Universal Robots PolyScope program: d02_cycle.urp

Program d02_cycle (installation=default directory=/programs createdIn=5.9.1.1031110 lastSavedIn=5.9.1.1031110 robotSerialNumber=20195501059)
Calibrated DH parameters: a=[0.000146, -0.418764, -0.053981, 0.000058, -0.000023, 0]; d=[0.162545, 37.319448, -206.067439, 168.881546, 0.09955, 0.099464]; alpha=[1.57004, -0.001979, 0.002304, 1.570607, -1.57066, 0]; deltaTheta=[0, -0.174616, -1.258233, 1.432844, -0.000001, 0]
BeforeStart
  URCap Gripper Activate (Robotiq_Grippers, Robotiq Inc.) dataModel(ResetAndActivateKey=false)
Robot Program (runOnlyOnce=true)
  Call d02_home
  Call d02_amp_off
  Call d02_unplug
  Call d02_replug
  Call d02_amp_on
  Call d02_home
SubProgram -> d02_home
SubProgram -> d02_amp_off
SubProgram -> d02_amp_on
SubProgram -> d02_unplug
SubProgram -> d02_replug
SubProgram d02_home (keepSynchronizedWithDisk=true) programFile=/programs/d02_home.urp
  URCap Gripper Activate (Robotiq_Grippers, Robotiq Inc.) dataModel(ResetAndActivateKey=false)
  URCap Gripper (Robotiq_Grippers, Robotiq Inc.) dataModel(position=65.0, force=100.0, speed=100.0, positionInDouble=65.0, forceInDouble=100.0, speedInDouble=100.0, slaveIds=[9], blocking=true)
  URCap Gripper (Robotiq_Grippers, Robotiq Inc.) dataModel(position=100.0, force=100.0, speed=100.0, positionInDouble=100.0, forceInDouble=100.0, speedInDouble=100.0, slaveIds=[9], blocking=false)
  MoveJ speed 60 deg/s, acceleration 80 deg/s^2 (useActiveTCP=true) feature=Base
    Waypoint Waypoint (Variable): variable(featureName=d02_home_p)
SubProgram d02_amp_off (keepSynchronizedWithDisk=true) programFile=/programs/d02_amp_off.urp
  URCap Gripper (Robotiq_Grippers, Robotiq Inc.) dataModel(position=100.0, force=100.0, speed=100.0, positionInDouble=100.0, forceInDouble=100.0, speedInDouble=100.0, slaveIds=[9], blocking=false)
  MoveL speed 250 mm/s, acceleration 1200 mm/s^2 (useActiveTCP=true) feature=Base
    Waypoint Waypoint (Variable): variable(featureName=d02_amp_sw_p)
    URCap Zero FT Sensor (Robotiq_Copilot, Robotiq Inc.) dataModel(NodeInitializedKey=true, WaitForSteadyWrenchOptionKey=true)
    URCap Force Control (Robotiq_Copilot, Robotiq Inc.) dataModel(NodeInitializedKey=true, force_x=0, force_y=0, force_mx=0, force_my=0, force_mz=0, limit_x_neg=-100, limit_y_neg=-100, limit_z_neg=-100, limit_x_pos=100, limit_y_pos=100, limit_z_pos=100, limit_mx_neg=-20, limit_my_neg=-20, limit_mz_neg=-20, limit_mx_pos=20, limit_my_pos=20, limit_mz_pos=20, ft_control_mx=false, ft_control_my=false, ft_control_mz=false, stiffness_x=100, stiffness_y=100, stiffness_z_position=100, stiffness_mx=100, stiffness_my=100, stiffness_mz=100, force_z=20, ft_control_y=false, ft_control_x=false, HackTriggeringContributionIsDefinedMethodKey=true, TranslatableFeatureKey=1, adaptive_stiffness=true, ft_control_z=true, is_force_control_about_actual_position=true)
      Wait Sleep waitTime=2
    Waypoint Waypoint (Variable): variable(featureName=d02_amp_sw_p)
SubProgram d02_unplug (keepSynchronizedWithDisk=true) programFile=/programs/d02_unplug.urp
  MoveL speed 250 mm/s, acceleration 1200 mm/s^2 (useActiveTCP=true) feature=Base
    Waypoint Waypoint (Variable): variable(featureName=d02_plug_p)
    URCap Gripper (Robotiq_Grippers, Robotiq Inc.) dataModel(position=100.0, force=100.0, speed=100.0, positionInDouble=100.0, forceInDouble=100.0, speedInDouble=100.0, slaveIds=[9], blocking=false)
    MoveDirectionNode (selectedDirection=ZPlus toolParams=0.02, 0.8) feature=Joint_6_name
      Until TOOL_CONTACT_DETECTION (allowActions=true retraction=0.001 decelerationAcceleration=3 decelerationAngularAcceleration=34.906585)
        URCap Gripper (Robotiq_Grippers, Robotiq Inc.) dataModel(position=65.0, force=100.0, speed=100.0, positionInDouble=65.0, forceInDouble=100.0, speedInDouble=100.0, slaveIds=[9], blocking=true)
        MoveDirectionNode (selectedDirection=ZPlus toolParams=0.05, 0.8) feature=Joint_6_name
          Until DISTANCE (allowActions=false deceleration=3 distanceNodeType=STOP) Distance=0.02; motionParameters(blendRadius=0)
        URCap Gripper (Robotiq_Grippers, Robotiq Inc.) dataModel(position=100.0, force=100.0, speed=100.0, positionInDouble=100.0, forceInDouble=100.0, speedInDouble=100.0, slaveIds=[9], blocking=true)
        MoveL speed 25 mm/s, acceleration 1200 mm/s^2 (useActiveTCP=true) feature=Base
          Waypoint Pull (Relative): relativeFromPosition TCP in base x=108.075 y=-582.031 z=19.139 mm, rx=-2.2457 ry=-2.1683 rz=0.0242 rad; joints [88.128, -64.848, 105.271, -130.26, 268.593, 90.173] deg; TCP offset x=0 y=0 z=174 mm, rx=0 ry=0 rz=0 rad; TCP in base x=109.536 y=-542.231 z=19.13 mm, rx=-2.2458 ry=-2.1682 rz=0.0241 rad; joints [88.149, -69.075, 111.89, -132.649, 268.605, 90.202] deg
      Until DISTANCE (allowActions=true deceleration=3 distanceNodeType=STOP) Distance=0.02; motionParameters(blendRadius=0)
        Waypoint Waypoint (Variable): variable(featureName=d02_plug_p)
SubProgram d02_replug (keepSynchronizedWithDisk=true) programFile=/programs/d02_replug.urp
  URCap Insertion (Robotiq_Copilot, Robotiq Inc.) dataModel(NodeInitializedKey=true)
    URCap Zero FT Sensor (Robotiq_Copilot, Robotiq Inc.) dataModel(NodeInitializedKey=true, WaitForSteadyWrenchOptionKey=false)
    URCap Linear (Robotiq_Copilot, Robotiq Inc.) dataModel(NodeInitializedKey=true, fb_exit_insertion=false, fb_max_distance=50.0, fb_speed=10.0, fb_force=40.0, fbDirection=X-); state(isChildrenLocked=true)
      URCap On error (Robotiq_Copilot, Robotiq Inc.)
        'Sequence if maximum distance is reached'
        Halt
    URCap Gripper (Robotiq_Grippers, Robotiq Inc.) dataModel(position=65.0, force=100.0, speed=100.0, positionInDouble=65.0, forceInDouble=100.0, speedInDouble=100.0, slaveIds=[9], blocking=true)
    MoveL speed 250 mm/s, acceleration 1200 mm/s^2 (useActiveTCP=true) feature=Base
      MoveDirectionNode (selectedDirection=ZMinus) feature=Joint_6_name
        Until DISTANCE (allowActions=false deceleration=3 distanceNodeType=STOP) Distance=0.025; motionParameters(blendRadius=0)
SubProgram d02_amp_on (keepSynchronizedWithDisk=true) programFile=/programs/d02_amp_on.urp
  URCap Gripper (Robotiq_Grippers, Robotiq Inc.) dataModel(position=100.0, force=100.0, speed=100.0, positionInDouble=100.0, forceInDouble=100.0, speedInDouble=100.0, slaveIds=[9], blocking=false)
  MoveL speed 250 mm/s, acceleration 1200 mm/s^2 (useActiveTCP=true) feature=Base
    Waypoint Waypoint (Variable): variable(featureName=d02_amp_sw_p)
    MoveDirectionNode (selectedDirection=ZPlus toolParams=0.01, 0.8) feature=Joint_6_name
      Until TOOL_CONTACT_DETECTION (allowActions=false retraction=0 decelerationAcceleration=3 decelerationAngularAcceleration=34.906585)
    URCap Gripper (Robotiq_Grippers, Robotiq Inc.) dataModel(position=75.29411764705883, force=100.0, speed=100.0, positionInDouble=75.29411764705883, forceInDouble=100.0, speedInDouble=100.0, slaveIds=[9], blocking=true)
    MoveDirectionNode (selectedDirection=ZPlus toolParams=0.01, 0.8) feature=Joint_6_name
      Until DISTANCE (allowActions=false deceleration=3 distanceNodeType=STOP) Distance=0.01; motionParameters(blendRadius=0)
    URCap Gripper (Robotiq_Grippers, Robotiq Inc.) dataModel(position=100.0, force=100.0, speed=100.0, positionInDouble=100.0, forceInDouble=100.0, speedInDouble=100.0, slaveIds=[9], blocking=true)
    URCap Force Control (Robotiq_Copilot, Robotiq Inc.) dataModel(NodeInitializedKey=true, force_x=0, force_y=0, force_mx=0, force_my=0, force_mz=0, limit_x_neg=-100, limit_y_neg=-100, limit_z_neg=-100, limit_x_pos=100, limit_y_pos=100, limit_z_pos=100, limit_mx_neg=-20, limit_my_neg=-20, limit_mz_neg=-20, limit_mx_pos=20, limit_my_pos=20, limit_mz_pos=20, ft_control_x=false, ft_control_y=false, ft_control_mx=false, ft_control_my=false, ft_control_mz=false, stiffness_x=100, stiffness_y=100, stiffness_z_position=100, stiffness_mx=100, stiffness_my=100, stiffness_mz=100, force_z=-15, adaptive_stiffness=true, ft_control_z=true, is_force_control_about_actual_position=true, TranslatableFeatureKey=1, HackTriggeringContributionIsDefinedMethodKey=true)
      Wait Sleep waitTime=2
      URCap Gripper (Robotiq_Grippers, Robotiq Inc.) dataModel(position=75.0, force=100.0, speed=100.0, positionInDouble=75.0, forceInDouble=100.0, speedInDouble=100.0, slaveIds=[9], blocking=true)
    Waypoint Waypoint (Variable): variable(featureName=d02_amp_sw_p)
